// alias for a state text for FB_StateMachine
TYPE
  A_StateText    : STRING[31];
END_TYPE

(* stored: Version 1.1.0.1, ProductVersion 3.1.4024.4
   DUT A_StateText: Id {102a4782-c208-4b33-ad3f-c509b67e0a38} *)
